(* PLC project BlogProject.project, CODESYS CODESYS V3.5 SP14 Patch 3 *)
(* stored: creationDateTime 2021-10-07T21:06:52.6289988, modificationDateTime 2021-10-07T20:40:20.1109198 *)

FUNCTION_BLOCK mcNoAction IMPLEMENTS itfAction

            
          

METHOD getAction : BOOL
                  
                
END_METHOD
END_FUNCTION_BLOCK
